Staubli VAL3: trackOffJ.pgx

public program trackOffJ(joint x_jLoc (dimensions=1), tool x_tTool (dimensions=1), mdesc x_mDesc (dimensions=1), num& x_nMoveID (dimensions=1), num& x_nError[] (dimensions=1))
// Perform motion to de-synchronize from conveyor to a joint location
  local num l_bLock
  local num l_nStep
begin
  // This program executes the motion to leave the conveyor
  //  to a joint location
  //
  // Input Param
  //  x_jLoc    : Joint location to reach
  //  x_tTool   : Tool for motion
  //  x_nMoveID : ID of the movement on the motion stack
  //  x_mDesc   : Motion descriptor
  //
  // Output Param
  //  x_nError : Error code
  //            = 0 : No error
  //            = 1 : No object ID selected
  //
  //----------------------------------------------------------------
  //
  x_nError=0
  // Check if the robot is synchronized (user must have invoked trackOn)
  if nMobFrameSync>=0
    tTool.trsf=position(x_tTool,flange)
    mTrackOff=x_mDesc
    if mTrackOff.blend==joint
      mTrackOff.blend=Cartesian
    endIf
    x_nMoveID=$trackOff(x_jLoc,x_tTool,mTrackOff)
    // Robot is not synchronized with any conveyor
    nMobFrameSync=-1
    //
    if bAnd(cfg:nLog,cfg:nLOGMOTION)==cfg:nLOGMOTION
      logMsg("MOT(trackOff)>>Request to desynchronize from conveyor"+toString("2",nCnvSynch))
    endIf
  else
    x_nError=1
    if cfg:bLog
      logMsg("MOT(trackOff)>>Robot is not synchronised with conveyor"+toString("2",nCnvSynch))
    endIf
  endIf
end
